(* LS Electric XG5000 project: 02_03_Practice1 *)
(* PLC LSPLC *)
(* module base 0 slot 0: 입력 모듈:XGI-D21A (DC 24V 입력, 8점 (전류소스/싱크입력)) *)
(* module base 0 slot 1: 출력 모듈:XGQ-RY1A (릴레이 출력, 8점 (2A용, 단독 COM.)) *)

(* Comments on direct variables
%IX0.0.0	P1
%IX0.0.1	P2
%QX0.1.0	P40
%QX0.1.1	P41
*)

PROGRAM NewProgram (* task: 스캔 프로그램 *)
VAR
    P1 AT %IX0.0.0 : BOOL; (* 입력 *)
    P2 AT %IX0.0.1 : BOOL; (* 입력 *)
    P40 AT %QX0.1.0 : BOOL; (* 출력 *)
    P41 AT %QX0.1.1 : BOOL; (* 출력 *)
END_VAR

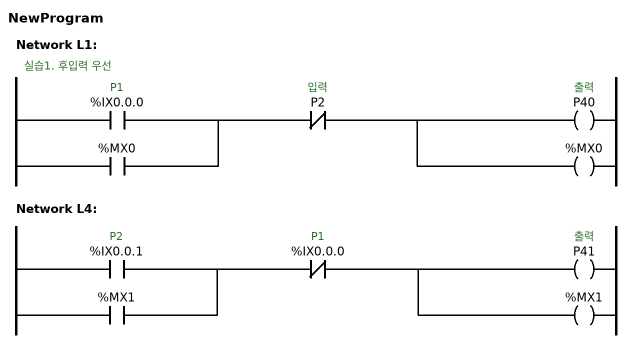
(* 실습1. 후입력 우선 *)
(* Rung L1 *)
P40 := (%IX0.0.0 OR %MX0) AND NOT P2;
%MX0 := (%IX0.0.0 OR %MX0) AND NOT P2;
(* Rung L4 *)
P41 := (%IX0.0.1 OR %MX1) AND NOT %IX0.0.0;
%MX1 := (%IX0.0.1 OR %MX1) AND NOT %IX0.0.0;
END_PROGRAM